PROGRAM MAIN
VAR
END_VAR

END_PROGRAM

(* stored: Version 1.1.0.1
   POU MAIN: Id {660e0362-f648-4dfc-847c-d52080f10f80} *)
